{attribute 'qualified_only'}
{attribute 'strict'}
{attribute 'to_string'}
TYPE E_RobotCommand :
(
    None := 0,
    Home := 1,
    MoveJoints := 2,
    MoveJointsRelative := 3,
    MovePose := 4,
    MoveLinear := 5,
    Stop := 6,
    Pause := 7,
    Resume := 8,
    SetSpeedOverride := 9,
    MoveLinearRelative := 10,
    SetDigitalOutput := 11,
	GoTo := 12
);
END_TYPE

(* stored: Version 1.1.0.1, ProductVersion 3.1.4026.18
   DUT E_RobotCommand: Id {0e6e3e13-8f2b-4379-9019-d5b4d0bf289c} *)
